FUNCTION_BLOCK MM540
VAR_INPUT
END_VAR
VAR_OUTPUT
	// 等待觸發中
	bActive : BOOL;
	// 忙碌中
	bBuzy : BOOL;
	// 已完成
	bDone : BOOL;
	// 發生錯誤
	bError : BOOL;
END_VAR
VAR
	FeedCar_Enc_raw : MM540_Raw;
	
	Step : INT;
	
	_SetPos : DINT;
	
	_timeout	: TIME := T#10S;
	
	_timeTmr	: TON;
END_VAR

bBuzy := Step > 0 AND Step < 10000;
bActive := FeedCar_Enc_raw.Inc_Preload_Trigger > 0 AND bBuzy;
bError := Step >= 10000;

CASE Step OF
	1000: // 相關暫存器復位
		FeedCar_Enc_raw.Inc_Preload_Trigger := 0;
		bDone := FALSE;
		bActive := TRUE;
		step := step + 1;
		
	1001:
		IF NOT FeedCar_Enc_raw.Inc_Preload_Done THEN
			step := step + 1;
		END_IF
		
	1002:
		step := 1010;
		
		
	1010: // 放置要設定的值
		FeedCar_Enc_raw.Inc_Preload_Value := _SetPos;
		step := step + 1;
		
	1011:
		FeedCar_Enc_raw.Inc_Preload_Trigger := 2;
		_timeTmr.IN := TRUE;
		step := step + 1;
		
	1012:
		IF FeedCar_Enc_raw.Inc_Preload_Done OR _timeTmr.Q THEN 
			
			FeedCar_Enc_raw.Inc_Preload_Trigger := 0;
			_timeTmr.IN := FALSE;
			bActive := FALSE;
			
			// 歸零完成
			IF FeedCar_Enc_raw.Inc_Preload_Done THEN
				step := 1020;
			// 歸零超時
			ELSIF _timeTmr.Q THEN
				step := 1050;
			END_IF
		END_IF
		
	1020:// 歸零完成
		bdone := TRUE;
		step := 0;
		
		
	1050: // 歸零超時
		step := 10000;
END_CASE



_timeTmr(PT:=_timeout);

PROPERTY Buzy : bool
GET
Buzy := bbuzy;
END_GET
END_PROPERTY

PROPERTY Done : bool
GET
Done := bdone;
END_GET
END_PROPERTY

PROPERTY Error : bool
GET
Error := bError;
END_GET
END_PROPERTY

PROPERTY Pos : REAL
GET
Pos := DINT_TO_REAL(FeedCar_Enc_raw.Inc);
END_GET
END_PROPERTY

METHOD SetPos : BOOL
VAR_INPUT
	Pos : DINT;
END_VAR
_SetPos := Pos;

step := 1000;
END_METHOD

END_FUNCTION_BLOCK

(* stored: Version 1.1.0.1, ProductVersion 3.1.4024.15
   POU MM540: Id {fed5345a-fcd3-40c6-97f5-f3301df14d6b}, SpecialFunc None
   Property Buzy: Id {0652a691-38e3-4da2-a9bb-b898d861b9a7}
   Get Get: Id {9761f28c-ae4d-4193-b22b-03fa4cb20d92}
   Property Done: Id {bb7e25aa-677b-433c-8a65-515338f716d4}
   Get Get: Id {fb14ae47-fbed-4c2b-a788-28fadbfa1c96}
   Property Error: Id {1eea8231-c8f7-46a6-a136-ab6e164ec389}
   Get Get: Id {3a8ab407-2ba2-4317-9c74-5ecc218570e2}
   Property Pos: Id {ce0e3907-5815-4eee-868e-643b65e33b82}
   Get Get: Id {5fd39996-d208-42e0-9e09-d2caedaebf49}
   Method SetPos: Id {1cda5e08-9bc3-47a2-9a0f-96fdb3aafa3b} *)
